{attribute 'GeneratedUsingTerminal: KL6401-0002'}
{attribute addProperty BoxType "KL6401-0002"}
{attribute addProperty Id "Channel_1AT %Q*Channel_7606D9890"}
{attribute addProperty CRC "2434187969"}
{attribute addProperty Size "0"}
TYPE KL_9116C2C1 :
STRUCT
	{attribute addProperty Name "Channel_1"}
	Channel_1 : Channel_7606D989;
END_STRUCT
END_TYPE

(* stored: Version 1.2.0.0, ProductVersion 3.1.4024.9
   DUT KL_9116C2C1: Id {8667008c-f867-4ec5-aba3-eb839ac96848} *)
